(* IEC 61131-3 sources: lc3-wifi-kurs/src/example_5_hysteresis, 1 file *)

(* ---- Program_Hysteresis.iecfbd ---- *)
PROGRAM Program_Hysteresis
  VAR
    i2c_handle : DINT := -1;
    analog_values : ARRAY[0..4] OF UINT;
    digital_values : ARRAY[0..7] OF BOOL;
    Schmitt_Trigger1 : Schmitt_Trigger;
  END_VAR
  VAR_OUTPUT
    digital_output : BOOL;
  END_VAR

  (*

    // Network 1:
    LT(IN1 := i2c_handle, IN2 := 0, LT => @C(22).LT);
    I2C_open(EN := @C(22).LT, bus_id := 1, I2C_open => i2c_handle);

    // Network 2:
    @VF(43) := I2C_ADDRESSES#I2HAE_1;
    GE(IN1 := i2c_handle, IN2 := 0, GE => @C(28).GE);
    I2C_I2HAE_read(EN := @C(28).GE, fd := i2c_handle, address := @VF(43), values => analog_values);

    // Network 3:
    Schmitt_Trigger1(in := analog_values[0], low := 300, high := 700);
    digital_values[0] := Schmitt_Trigger1.out;

    // Network 4:
    @VF(41) := I2C_ADDRESSES#PCF8574_OUTPUT_1;
    GE(IN1 := i2c_handle, IN2 := 0, GE => @C(45).GE);
    I2C_PCF8574_write(EN := @C(45).GE, fd := i2c_handle, address := @VF(41), pin_values := digital_values);

  *)

  @VF(9) : @E(300), @R(99.9, 560.0, 140.0, 19.0), DINT;
  @VF(10) : @E(700), @R(99.9, 579.6, 140.0, 19.0), DINT;
  @VF(16) : @E(i2c_handle), @R(90.0, 300.0, 140.0, 19.0);
  @C(18) : @F(I2C_open), @R(487.8, 190.0, 160.0, 38.5), @I(@N(EN), @L(9.5)), @I(@N(bus_id), @L(29.5)), @O(@N(ENO), @R(9.5)), @O(@N(I2C_open), @R(29.5));
  @VF(21) : @E(i2c_handle), @R(89.7, 100.4, 140.0, 19.0);
  @C(22) : @F(LT), @R(269.7, 100.4, 40.0, 38.0), DINT, @I(@N(IN1), @L(9.5)), @I(@N(IN2), @L(29.5)), @O(@N(LT), @R(9.5));
  @VF(23) : @E(0), @R(89.7, 120.4, 140.0, 19.0), DINT;
  @VF(17) : @E(i2c_handle), @R(750.0, 210.0, 140.0, 19.0);
  @C(28) : @F(GE), @R(340.2, 299.5, 40.0, 38.0), DINT, @I(@N(IN1), @L(9.5)), @I(@N(IN2), @L(29.5)), @O(@N(GE), @R(9.5));
  @VF(31) : @E(0), @R(90.0, 320.0, 140.0, 19.0), DINT;
  @C(29) : @F(I2C_I2HAE_read), @R(490.0, 320.0, 150.0, 140.0), @I(@N(EN), @L(9.5)), @I(@N(fd), @L(29.5)), @I(@N(address), @L(49.5)), @O(@N(ENO), @R(9.5)), @O(@N(values), @R(29.5));
  @VF(1) : @E(analog_values), @R(750.0, 340.0, 140.0, 19.0);
  @VF(37) : @E(analog_values[0]), @R(99.9, 540.0, 170.0, 19.0);
  @C(38) : @F(I2C_PCF8574_write), @R(510.0, 830.0, 160.0, 88.0), @I(@N(EN), @L(19.5)), @I(@N(fd), @L(39.5)), @I(@N(address), @L(59.5)), @I(@N(pin_values), @L(79.5)), @O(@N(ENO), @R(19.5));
  @VF(39) : @E(digital_values[0]), @R(750.0, 540.0, 170.0, 19.0);
  @VF(4) : @E(digital_values), @R(110.0, 900.0, 140.0, 19.0);
  @VF(41) : @E(I2C_ADDRESSES#PCF8574_OUTPUT_1), @R(110.0, 880.0, 140.0, 19.0);
  @VF(43) : @E(I2C_ADDRESSES#I2HAE_1), @R(90.0, 360.0, 140.0, 19.0);
  @VF(35) : @E(i2c_handle), @R(110.0, 860.0, 140.0, 19.0);
  @C(45) : @F(GE), @R(360.0, 820.0, 40.0, 38.0), DINT, @I(@N(IN1), @L(9.5)), @I(@N(IN2), @L(29.5)), @O(@N(GE), @R(9.5));
  @VF(46) : @E(0), @R(110.0, 840.0, 140.0, 19.0), DINT;
  @VF(19) : @E(1), @R(90.0, 210.0, 140.0, 19.0), INT;
  @C(3) : @FB(Schmitt_Trigger1), @R(460.0, 540.0, 120.0, 160.0), @I(@N(in), @L(9.5)), @I(@N(low), @L(29.5)), @I(@N(high), @L(49.5)), @O(@N(out), @R(9.5));
  @CP(33) : 251.0, 309.5;
  @CP(48) : 292.6, 869.5;

  @G(24) :
     @L(@VF(23).o, @C(22).IN2)
    ;
  @G(25) :
     @L(@VF(21).o, @C(22).IN1)
    ;
  @G(26) :
     @L(@C(22).LT, @C(18).EN)
    ;
  @G(27) :
     @L(@C(18).I2C_open, @VF(17).i)
    ;
  @G(30) :
     @L(@VF(16).o, @CP(33)),
     @L(@CP(33), @C(28).IN1),
     @L(@CP(33), @C(29).fd)
    ;
  @G(32) :
     @L(@VF(31).o, @C(28).IN2)
    ;
  @G(15) :
     @L(@C(28).GE, @C(29).EN)
    ;
  @G(36) :
     @L(@C(29).values, @VF(1).i)
    ;
  @G(40) :
     @L(@VF(4).o, @C(38).pin_values)
    ;
  @G(42) :
     @L(@VF(41).o, @C(38).address)
    ;
  @G(34) :
     @L(@VF(43).o, @C(29).address)
    ;
  @G(44) :
     @L(@VF(35).o, @CP(48)),
     @L(@CP(48), @C(38).fd),
     @L(@CP(48), @C(45).IN1)
    ;
  @G(47) :
     @L(@VF(46).o, @C(45).IN2)
    ;
  @G(49) :
     @L(@C(45).GE, @C(38).EN)
    ;
  @G(20) :
     @L(@VF(19).o, @C(18).bus_id)
    ;
  @G(2) :
     @L(@VF(37).o, @C(3).in)
    ;
  @G(5) :
     @L(@VF(9).o, @C(3).low)
    ;
  @G(6) :
     @L(@VF(10).o, @C(3).high)
    ;
  @G(7) :
     @L(@C(3).out, @VF(39).i)
    ;
END_PROGRAM
